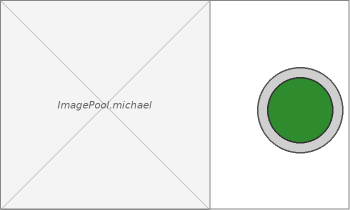
VISUALIZATION VISU_Run  // 350x210
    Lamp1 (250,60 100x100), variable: GVL.bRunLamp, style: Lamp-Lamp1-Green
    Image (11,118 150x30), image: ImagePool.homeButton
    Image (0,0 210x210), image: ImagePool.michael
        p84334746: GVL.sImage
        OnMouseClick: toggle bRun
END_VISUALIZATION

(* stored: Version 1.1.0.1
   Visu VISU_Run: Id {a84c4134-e2bf-49bf-bd47-cd98a3f16397} *)
